FUNCTION_BLOCK TAdsWrite
VAR
    Execution : TExecution;
    AdsWrite1 : ADSWRITE := (TMOUT := T#2S);
END_VAR

AdsWrite1(
	NETID:= , 
	PORT:= , 
	IDXGRP:= , 
	IDXOFFS:= , 
	LEN:= , 
	SRCADDR:= , 
	WRITE:= Execution.Starting, 
	TMOUT:= , 
	BUSY=> , 
	ERR=> , 
	ERRID=> );
    
IF Execution.Starting THEN
    Execution.SetBusy();
END_IF
IF Execution.Busy AND NOT AdsWrite1.BUSY THEN
    IF AdsWrite1.ERR THEN
        Execution.SetError(AdsWrite1.ERRID);
    ELSE
        Execution.SetDone();
	END_IF
END_IF

METHOD Execute : BOOL
VAR_INPUT
	AmsNetId:T_AmsNetid;
	Port:T_AmsPort;
	IndexGroup:UDINT; 
	IndexOffset:UDINT;
	DataLength:UDINT; 
	DataAddress:PVOID; 
END_VAR
AdsWrite1.NETID := AmsNetId;
AdsWrite1.PORT := Port;
AdsWrite1.IDXGRP := IndexGroup;
AdsWrite1.IDXOFFS := IndexOffset;
AdsWrite1.LEN := DataLength;
AdsWrite1.SRCADDR := DataAddress;
Execute := Execution.Start();
END_METHOD

PROPERTY ExecutionResult : IExecutionResult
GET
ExecutionResult := Execution;
END_GET
END_PROPERTY

END_FUNCTION_BLOCK

(* stored: Version 1.1.0.1, ProductVersion 3.1.4022.12
   POU TAdsWrite: Id {0518a10c-18cf-4c41-b7e4-3dad0dec5061}, SpecialFunc None
   Method Execute: Id {10b24599-5f24-46a2-8e4d-3e8c401c8032}
   Property ExecutionResult: Id {587b581d-2649-48ad-b252-d24722c9f199}
   Get Get: Id {2af0530e-1a27-472a-aea5-27a80db99102} *)
